PROGRAM main
VAR
	MODBEE_HW_INPUTS0 : MODBEE_HW_INPUTS;
	MODBEE_HW_OUTPUTS0 : MODBEE_HW_OUTPUTS;
	start : bool;
	stop : bool;
	run : bool;
END_VAR

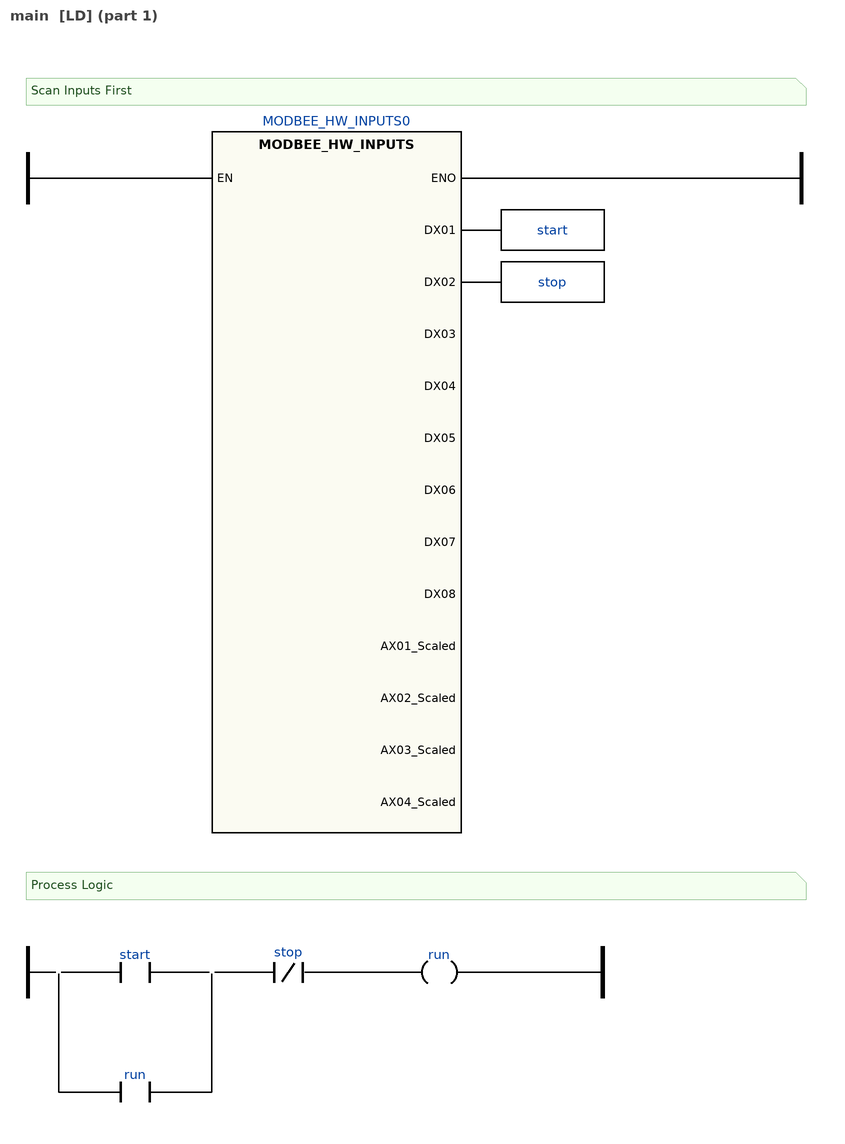
(* LD diagram, written out as Structured Text *)
(* Scan Inputs First *)
MODBEE_HW_INPUTS0();
start := MODBEE_HW_INPUTS0.DX01;
stop := MODBEE_HW_INPUTS0.DX02;
(* Process Logic *)
run := (run OR start) AND NOT stop;
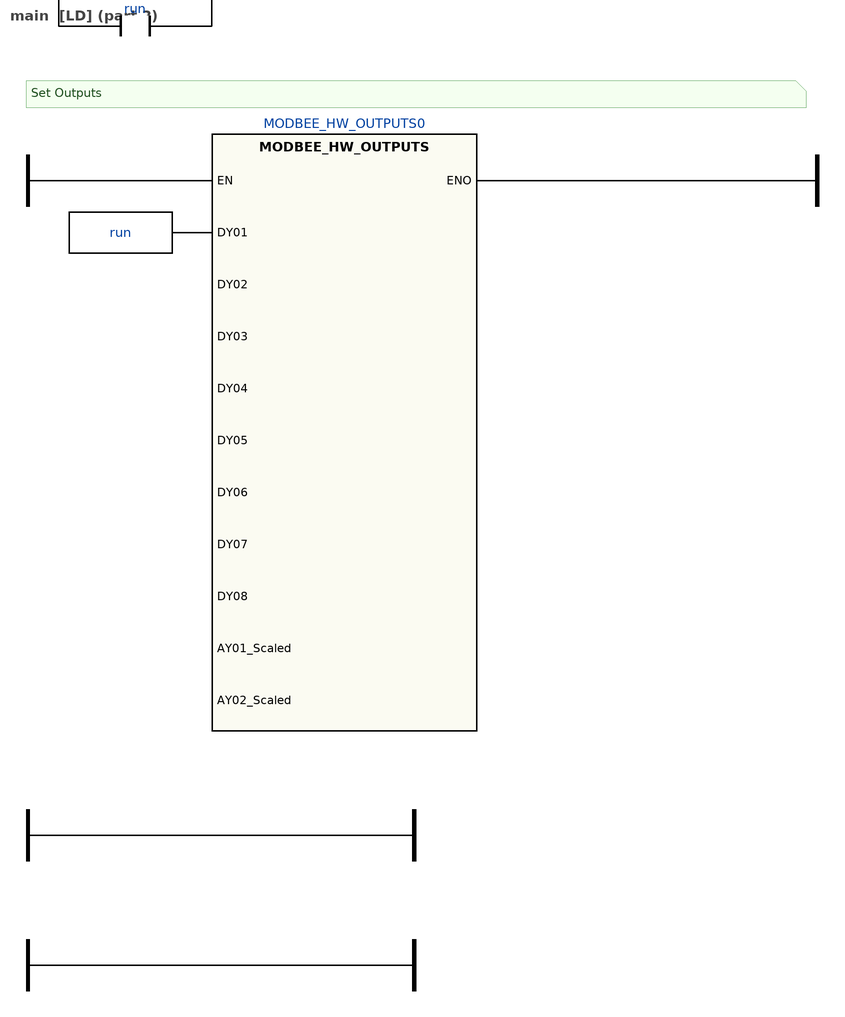
(* Set Outputs *)
MODBEE_HW_OUTPUTS0(DY01 := run);
END_PROGRAM
